ABB RobotStudio station: Proyecto_PRR.rsstnx

Station Proyecto_PRR (saved by RobotStudio 23.2.10395.0)
Layout (positions relative to the parent item):
  - IRB920T_6_55_30_R_02 [mechanism, from %ABB.RobotStudio.Models.IRB920%\IRB920T_6_55_30_R_02.rslib] at (-1.39, 0, 835) mm, rotated rx 0 ry 0 rz 90 deg; joint values [0, 0.2618, -0.01, 0] (rad or m)
  - Mi_Ventosa_3 [smart component, from Libraries\1217c23c-7d3e-48fb-b7d3-d1b2005a3c2bMi_Ventosa.rslib] at (-68.68, 541.14, 1026.5) mm, rotated rx 180 ry 0 rz 105 deg
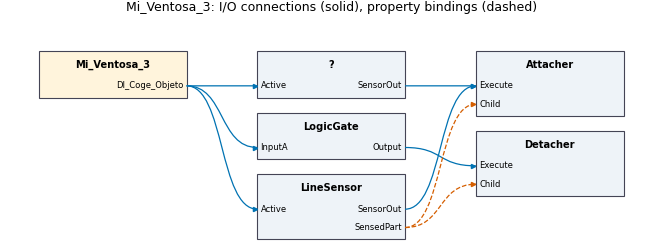
      connections:
        Mi_Ventosa_3.DI_Coge_Objeto -> ?.Active
        ?.SensorOut -> Attacher.Execute
        Mi_Ventosa_3.DI_Coge_Objeto -> LogicGate.InputA
        LogicGate.Output -> Detacher.Execute
        Mi_Ventosa_3.DI_Coge_Objeto -> LineSensor.Active
        LineSensor.SensorOut -> Attacher.Execute
        LineSensor.SensedPart => Attacher.Child
        LineSensor.SensedPart => Detacher.Child
    - Attacher [smart component, from Components\Attacher.rslib]
        properties: Parent=Ventosa; Flange=0; Child=(none); Mount=false; Offset=[0 0 0]; Orientation=[0 0 0]
    - Detacher [smart component, from Components\Detacher.rslib]
        properties: Child=(none); KeepPosition=true
    - Ventosa [mechanism, from Libraries\1217c23c-7d3e-48fb-b7d3-d1b2005a3c2bMi_Ventosa.rslib] at (0, 0, 0) mm
    - LogicGate [smart component, from Components\LogicGate.rslib]
        properties: Operator=NOT; Delay=0
    - LineSensor [smart component, from Components\LineSensor.rslib]
        properties: Start=[0 0 0.055]; End=[0 0 0.07]; Radius=0.001; SensedPart=(none); SensedPoint=[0 0 0]; Length=0.015; Tag=(none)
      - _sensorPart_ [part], size 2 x 2 x 15 mm
    - Indicador [part, from Libraries\1217c23c-7d3e-48fb-b7d3-d1b2005a3c2bMi_Ventosa.rslib] at (-4.38, 0, 0) mm
  - Conveyor [graphiccomponentgroup] at (-950, 1250, 0) mm
    - conveyorbelt-1kr - belt-1kr-1_2 [part] at (0, 0, 0) mm, rotated rx 90 ry 0 rz 0 deg, size 180 x 80 x 1996 mm
    - conveyorbelt-1kr - conv1-1kr-1_2 [part] at (0, 0, 0) mm, rotated rx 90 ry 0 rz 0 deg, size 50 x 100 x 2000 mm
    - conveyorbelt-1kr - conv1-1kr-2_2 [part] at (0, 0, 0) mm, rotated rx 90 ry 0 rz 0 deg, size 50 x 100 x 2000 mm
    - conveyorbelt-1kr - convsupp-1kr-1_2 [part] at (0, 0, 0) mm, rotated rx 90 ry 0 rz 0 deg, size 300 x 558.2 x 2000.5 mm
    - conveyorbelt-1kr - leg-1kr-1_2 [part] at (0, 0, 0) mm, rotated rx 90 ry 0 rz 0 deg, size 80 x 80 x 79.9 mm
    - conveyorbelt-1kr - leg-1kr-2_2 [part] at (0, 0, 0) mm, rotated rx 90 ry 0 rz 0 deg, size 80 x 80 x 79.9 mm
    - conveyorbelt-1kr - leg-1kr-3_2 [part] at (0, 0, 0) mm, rotated rx 90 ry 0 rz 0 deg, size 80 x 80 x 79.9 mm
    - conveyorbelt-1kr - leg-1kr-4_2 [part] at (0, 0, 0) mm, rotated rx 90 ry 0 rz 0 deg, size 80 x 80 x 79.9 mm
    - conveyorbelt-1kr - leg-1kr-15_2 [part] at (0, 0, 0) mm, rotated rx 90 ry 0 rz 0 deg, size 80 x 80 x 79.9 mm
    - conveyorbelt-1kr - leg-1kr-20_2 [part] at (0, 0, 0) mm, rotated rx 90 ry 0 rz 0 deg, size 80 x 80 x 79.9 mm
    - conveyorbelt-1kr - Part16-1kr-1_2 [part] at (0, 0, 0) mm, rotated rx 90 ry 0 rz 0 deg, size 200 x 30 x 30 mm
    - conveyorbelt-1kr - Part16-1kr-2_2 [part] at (0, 0, 0) mm, rotated rx 90 ry 0 rz 0 deg, size 200 x 30 x 30 mm
  - Conveyor_2 [graphiccomponentgroup] at (-125, 1250, 0) mm
    - conveyorbelt-1kr - belt-1kr-1_2 [part] at (0, 0, 0) mm, rotated rx 90 ry 0 rz 0 deg, size 180 x 80 x 1996 mm
    - conveyorbelt-1kr - conv1-1kr-1_2 [part] at (0, 0, 0) mm, rotated rx 90 ry 0 rz 0 deg, size 50 x 100 x 2000 mm
    - conveyorbelt-1kr - conv1-1kr-2_2 [part] at (0, 0, 0) mm, rotated rx 90 ry 0 rz 0 deg, size 50 x 100 x 2000 mm
    - conveyorbelt-1kr - convsupp-1kr-1_2 [part] at (0, 0, 0) mm, rotated rx 90 ry 0 rz 0 deg, size 300 x 558.2 x 2000.5 mm
    - conveyorbelt-1kr - leg-1kr-1_2 [part] at (0, 0, 0) mm, rotated rx 90 ry 0 rz 0 deg, size 80 x 80 x 79.9 mm
    - conveyorbelt-1kr - leg-1kr-2_2 [part] at (0, 0, 0) mm, rotated rx 90 ry 0 rz 0 deg, size 80 x 80 x 79.9 mm
    - conveyorbelt-1kr - leg-1kr-3_2 [part] at (0, 0, 0) mm, rotated rx 90 ry 0 rz 0 deg, size 80 x 80 x 79.9 mm
    - conveyorbelt-1kr - leg-1kr-4_2 [part] at (0, 0, 0) mm, rotated rx 90 ry 0 rz 0 deg, size 80 x 80 x 79.9 mm
    - conveyorbelt-1kr - leg-1kr-15_2 [part] at (0, 0, 0) mm, rotated rx 90 ry 0 rz 0 deg, size 80 x 80 x 79.9 mm
    - conveyorbelt-1kr - leg-1kr-20_2 [part] at (0, 0, 0) mm, rotated rx 90 ry 0 rz 0 deg, size 80 x 80 x 79.9 mm
    - conveyorbelt-1kr - Part16-1kr-1_2 [part] at (0, 0, 0) mm, rotated rx 90 ry 0 rz 0 deg, size 200 x 30 x 30 mm
    - conveyorbelt-1kr - Part16-1kr-2_2 [part] at (0, 0, 0) mm, rotated rx 90 ry 0 rz 0 deg, size 200 x 30 x 30 mm
  - 400_guide [part, from %ABB.RobotStudio.Models.Conveyors%\Conveyor Guide 400.rslib] at (198.86, 350, 0) mm, rotated rx 0 ry 0 rz 90 deg
  - tupperware [part] at (-69.33, 2180.39, 778.65) mm, rotated rx 90 ry 0 rz 0 deg, size 149.6 x 60.4 x 149.6 mm
  - tupperwarecap [part] at (-75.49, 2356.37, 779.72) mm, rotated rx 90 ry 0 rz 0 deg, size 151.2 x 15.2 x 163.2 mm
  - SoporteRobots [part] at (-146.31, -154.81, 0) mm, rotated rx 90 ry 0 rz 90 deg, size 287.2 x 850 x 287.2 mm
  - Pieza_4 [part] at (-125, 257.76, -23.11) mm, size 131.3 x 274 x 30 mm
  - Pieza_6 [part] at (115, 254.29, 6.52) mm, size 131.3 x 274 x 30 mm
  - Pieza_8 [part] at (-124.44, 0, -22.45) mm, size 5 x 257 x 30 mm
  - Pieza_9 [part] at (-285.02, 0, -22.45) mm, size 5 x 257 x 30 mm
Attachment: Mi_Ventosa_3 is attached to IRB920T_6_55_30_R_02 / Link4
Targets, tools, work objects and paths stored in the station, written as RAPID:
! task (no controller)
MODULE CalibData
  PERS tooldata TCP_Ventosa:=[TRUE,[[0,0,60],[1,0,0,0]],[0.1,[0,0,1],[1,0,0,0],0,0,0]];
ENDMODULE

